FUNCTION_BLOCK FB_PalletCheckAddonEmulation EXTENDS FB_FunctionConvEmulation
VAR_INPUT
END_VAR
VAR_OUTPUT
END_VAR
VAR
	pFunction						: POINTER TO FB_PalletCheckAddon; // Address to function
	rFunction						: REFERENCE TO FB_PalletCheckAddon; // Reference to function	
END_VAR

(**************************************************************************************************************
   Initialization
***************************************************************************************************************)
A_Init();


(**************************************************************************************************************
   Update reference
***************************************************************************************************************)
A_UpdateReference();

(**************************************************************************************************************
   Emulation
***************************************************************************************************************)
// If emulation function is initialized
IF FunctionData.Init THEN

	// Update data of real object
	M_UpdateRealObjectData();
		
	// Overwrite inputs	
	_M_OverWriteInputs();
END_IF

METHOD PRIVATE _M_OverWriteInputs
VAR_INPUT
END_VAR

VAR	
	
END_VAR

VAR_INST
	EmuState						: INT;
END_VAR

(**************************************************************************************
 * 	NAME		A_OverWriteInputs
 * 	FUNCTION	Overwrite inputs for emulation
 **************************************************************************************)

CASE EmuState OF
	0:
		rFunction.HW_Inputs.Sensor_RunnerTunnel := FALSE;
		rFunction.HW_Inputs.Sensor_TriggerStart  := FALSE;
		rFunction.HW_Inputs.Sensor_TriggerStop := FALSE;
		
		IF(rFunction._Trigger) THEN
			EmuState := EmuState+1;
		END_IF
		
	1,2,3,4,5,6,7,8,9:
		//give the real addon some time to execute
		EmuState := EmuState+1;
	
	10:
		//emulate TU reaching trigger start
		rFunction.HW_Inputs.Sensor_TriggerStart  := TRUE;
		rFunction.HW_Inputs.Sensor_RunnerTunnel := TRUE;
		EmuState := EmuState+1;
	11:
		rFunction.HW_Inputs.Sensor_TriggerStop := TRUE;
		EmuState := EmuState+1;
	
	12:
		IF(NOT rFunction._Trigger) THEN
			EmuState := EmuState+1;
		END_IF
	13:
		//done
		EmuState:=0;
		
	ELSE
		EmuState := 0;		
		
END_CASE

rFunction.HW_Inputs.Sensor_RunnerTunnel := rFunction.Config.HW_InputInverted.Sensor_RunnerTunnel XOR rFunction.HW_Inputs.Sensor_RunnerTunnel;
rFunction.HW_Inputs.Sensor_TriggerStart := rFunction.Config.HW_InputInverted.Sensor_TriggerStart XOR rFunction.HW_Inputs.Sensor_TriggerStart;
rFunction.HW_Inputs.Sensor_TriggerStop := rFunction.Config.HW_InputInverted.Sensor_TriggerStop XOR rFunction.HW_Inputs.Sensor_TriggerStop;
END_METHOD

ACTION A_Init:
(**************************************************************************************
 * 	NAME		A_Init
 * 	FUNCTION	Initialize emulated dummy function
 **************************************************************************************)

// If dummy function is not initialized
IF NOT FunctionData.Init Then
	// Check that linked dummy function number is valid
	IF eFunctionNumber > E_FunctionNumber.F_BEGIN_FUNCTION AND
	   eFunctionNumber < E_FunctionNumber.F_END_FUNCTION THEN   
		
		// Check if the real module is initialized
		IF F_IsFunctionInitialized(eFunctionNumber := eFunctionNumber) THEN
			// Module is initialized
			FunctionData.Init:= TRUE;
			
			// Send debug message
			DebugMsg := CONCAT('Initialization done. Element Function: ', FunctionRegistry[eFunctionNumber].FunctionName);
			fbDebugMsg.M_SendInfoMsg(DebugMsg);
			
			// Initialize real module
			F_InitializeFunction(eFunctionNumber := eFunctionNumber);
		END_IF
	END_IF
END_IF
END_ACTION

ACTION A_UpdateReference:
(**************************************************************************************
 * 	NAME		A_UpdateReference
 * 	FUNCTION	Update reference to real object
 **************************************************************************************)

// Check valid function number
IF eFunctionNumber > E_FunctionNumber.F_BEGIN_FUNCTION AND
   eFunctionNumber < E_FunctionNumber.F_END_FUNCTION THEN

	// Is reference valid  
	IF __ISVALIDREF(FunctionRegistry[eFunctionNumber].rFunction) THEN
		// Build address to reference
		pFunction := ADR(FunctionRegistry[eFunctionNumber].rFunction);

		// If address is possible
		IF pFunction <> 0 THEN
			// Build reference to memory
			rFunction REF= pFunction^;
		ELSE
			// Reinitialize module
			FunctionData.Init:= FALSE;
		END_IF
	ELSE
		// Reinitialize module
		FunctionData.Init:= FALSE;
	END_IF
END_IF
END_ACTION

END_FUNCTION_BLOCK

(* stored: Version 1.1.0.1, ProductVersion 3.1.4024.9
   POU FB_PalletCheckAddonEmulation: Id {81906258-d815-49e9-9f98-921af527c65d}, SpecialFunc None
   Method _M_OverWriteInputs: Id {0fb28ba9-ae88-4745-93e8-907469db019e}
   Action A_Init: Id {e0c8366e-871c-42d9-b74f-fe834b548fe7}
   Action A_UpdateReference: Id {387d7454-fb27-46b6-8fb6-900f076ce8cf} *)
